INTERFACE I_PersistentEventStorage

METHOD storeEvent
VAR_INPUT
	stEvent : ST_Event;
END_VAR
END_METHOD

END_INTERFACE

(* stored: Version 1.1.0.1, ProductVersion 3.1.4024.16
   Itf I_PersistentEventStorage: Id {ae09d5d4-c52b-4dab-8eff-230746920cf2}
   Method storeEvent: Id {3a7f4e83-f737-4ff9-91dd-35d6ca87b2cc} *)
